{attribute 'linkalways'}
{attribute 'no_explicit_call' := 'do not call this POU directly'}
FUNCTION_BLOCK Queue
VAR
	head : I_QueueNode;
END_VAR

METHOD PUBLIC Clear
VAR_INPUT
END_VAR
VAR
	current, next : I_QueueNode;
END_VAR
IF head = 0 THEN	
	RETURN;
END_IF

current := head; 

WHILE current.Next <> 0 DO
	next := current.next; 
	current.Destroy();
	current := next;
END_WHILE;
	
current.Destroy();
END_METHOD

METHOD FB_exit : BOOL
VAR_INPUT
	bInCopyCode : BOOL; // if TRUE, the exit method is called for exiting an instance that is copied afterwards (online change).
END_VAR
IF bInCopyCode THEN
	RETURN;
END_IF

Clear();
END_METHOD

METHOD PUBLIC Pop : BOOL;
VAR_INPUT
	Destination : ANY;
END_VAR
VAR
	transform : FB_JsonReadWriteDataType;
	next : I_QueueNode;
END_VAR
IF head = 0 THEN
	RETURN;
END_IF

IF head.DataType <> transform.GetDataTypeNameByAddress(Destination.diSize,Destination.pValue) THEN
	RETURN;
END_IF

next := head.Next;

Pop := head.Get(Destination);
head.Destroy();
head := next;
END_METHOD

METHOD PUBLIC Push
VAR_INPUT
	Item : ANY;
END_VAR
VAR
	pQueueNode : POINTER TO QueueNode;
	last : I_QueueNode;
END_VAR
pQueueNode := __NEW(QueueNode(Source := Item)); 

IF head = 0 THEN	
	head := pQueueNode^; 
	RETURN;
END_IF

last := head; 

WHILE last.Next <> 0 DO
	last := last.next; 
END_WHILE;
	
last.next := pQueueNode^;
END_METHOD

METHOD PUBLIC Size : UINT
VAR
	currentCount : UINT;
	currentNode : I_QueueNode;
END_VAR
currentCount := 0;
currentNode := head;

WHILE currentNode <> 0 DO
	currentNode := currentNode.Next;
	currentCount := currentCount + 1;
END_WHILE;

Size := currentCount;
END_METHOD

END_FUNCTION_BLOCK

(* stored: Version 1.1.0.1, ProductVersion 3.1.4024.11
   POU Queue: Id {1560f4e8-0d30-4cd0-8a35-4cb789c690a0}, SpecialFunc None
   Folder Destructor: Id {07801cfe-e9f1-4f70-9193-b414630971ad}
   Method Clear: Id {ceb7ff56-02be-4942-a18b-24e6bdf422bf}
   Method FB_exit: Id {d3f33f7d-ac2f-4275-af05-b8ab00d9c89d}
   Method Pop: Id {1ebc705c-ca50-401d-8bfc-812a17ac732a}
   Method Push: Id {5f56d2fb-90cb-4948-8ebe-7045801f934b}
   Method Size: Id {80cdf951-b102-45e6-9833-c35c6ce7d613} *)
